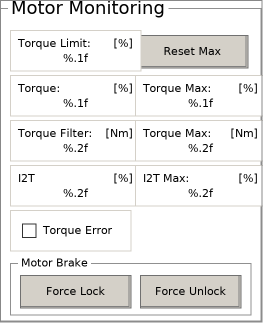
VISUALIZATION PH_MotorMonitoring  // 263x323
//==================================================================================================
//							Beckhoff Automation Poland
//									18.04.2018
//	Wizualizacja dla Axis Online
//  v1.0	|| TC v 3.1.4022.16		|| - pierwsza wersja
//==================================================================================================
VAR_IN_OUT
	stMcAxisOnline			: ST_McAxisOnline;	
END_VAR
    Rectangle (0,12 261x308)
    GroupBox (0,0 261x321), "Motor Monitoring"
        Button (137,35 111x33), "Reset Max"
            tap stMcAxisOnline.stMotorMonitoring.bReset
        Group (10,30 121x41)
            Textfield (0,0 131x41)
            Textfield (5,5 116x17), "Torque Limit:"
            Textfield (5,20 121x17), "%.1f", text variable: stMcAxisOnline.stMotorMonitoring.rTorqueLimit
            Textfield (85,5 41x17), "[%]"
        Group (10,75 121x41)
            Textfield (0,0 131x41)
            Textfield (5,5 116x17), "Torque:"
            Textfield (5,20 121x17), "%.1f", text variable: stMcAxisOnline.stMotorMonitoring.rTorquePerc
            Textfield (85,5 41x17), "[%]"
        Group (135,75 116x41)
            Textfield (0,0 131x41)
            Textfield (5,5 116x17), "Torque Max:"
            Textfield (5,20 121x17), "%.1f", text variable: stMcAxisOnline.stMotorMonitoring.rTorquePercMax
            Textfield (85,5 41x17), "[%]"
        Group (10,120 121x41)
            Textfield (0,0 131x41)
            Textfield (5,5 116x17), "Torque Filter:"
            Textfield (5,20 121x17), "%.2f", text variable: stMcAxisOnline.stMotorMonitoring.rTorqueF
            Textfield (85,5 41x17), "[Nm]"
        Group (135,120 116x41)
            Textfield (0,0 131x41)
            Textfield (5,5 116x17), "Torque Max:"
            Textfield (5,20 121x17), "%.2f", text variable: stMcAxisOnline.stMotorMonitoring.rTorqueMax
            Textfield (85,5 41x17), "[Nm]"
        Group (10,165 121x41)
            Textfield (0,0 131x41)
            Textfield (5,5 116x17), "I2T"
            Textfield (5,20 121x17), "%.2f", text variable: stMcAxisOnline.stMotorMonitoring.rI2T
            Textfield (85,5 41x17), "[%]"
        Group (135,165 116x41)
            Textfield (0,0 131x41)
            Textfield (5,5 116x17), "I2T Max:"
            Textfield (5,20 121x17), "%.2f", text variable: stMcAxisOnline.stMotorMonitoring.rI2TMax
            Textfield (85,5 41x17), "[%]"
        Group (10,210 121x41)
            Textfield (0,0 121x41), colour toggle: stMcAxisOnline.stMotorMonitoring.bError
            Checkbox (10,10 102x21), "Torque Error", variable: stMcAxisOnline.stStatus.stAxisStatus.NotMoving
        GroupBox (10,255 241x60), "Motor Brake"
            Button (130,20 101x33), "Force Unlock"
                tap stMcAxisOnline.stHoldingBrake.bForceUnlock
            Button (10,20 111x33), "Force Lock"
                tap stMcAxisOnline.stHoldingBrake.bForceLock
END_VISUALIZATION

(* stored: Version 1.1.0.1, ProductVersion 3.1.4026.12
   Visu PH_MotorMonitoring: Id {c8df21a5-14f0-454a-9e49-5662c6056221} *)
